{attribute 'GeneratedUsingTerminal: EP2339-0021-0016'}
{attribute addProperty BoxType "EP2339-0021-0016"}
{attribute addProperty Id "Channel_1AT %I*Channel_830843C11Channel_2AT %I*Channel_830843C11Channel_3AT %I*Channel_830843C11Channel_4AT %I*Channel_830843C11Channel_5AT %I*Channel_830843C11Channel_6AT %I*Channel_830843C11Channel_7AT %I*Channel_830843C11Channel_8AT %I*Channel_830843C11Channel_9AT %I*Channel_830843C11Channel_10AT %I*Channel_830843C11Channel_11AT %I*Channel_830843C11Channel_12AT %I*Channel_830843C11Channel_13AT %I*Channel_830843C11Channel_14AT %I*Channel_830843C11Channel_15AT %I*Channel_830843C11Channel_16AT %I*Channel_830843C11Channel_1_1AT %Q*Channel_42CA91F71Channel_2_1AT %Q*Channel_42CA91F71Channel_3_1AT %Q*Channel_42CA91F71Channel_4_1AT %Q*Channel_42CA91F71Channel_5_1AT %Q*Channel_42CA91F71Channel_6_1AT %Q*Channel_42CA91F71Channel_7_1AT %Q*Channel_42CA91F71Channel_8_1AT %Q*Channel_42CA91F71Channel_9_1AT %Q*Channel_42CA91F71Channel_10_1AT %Q*Channel_42CA91F71Channel_11_1AT %Q*Channel_42CA91F71Channel_12_1AT %Q*Channel_42CA91F71Channel_13_1AT %Q*Channel_42CA91F71Channel_14_1AT %Q*Channel_42CA91F71Channel_15_1AT %Q*Channel_42CA91F71Channel_16_1AT %Q*Channel_42CA91F71WcStateAT %I*WcState_9091E0EB2InfoDataAT %I*InfoData_07DD5D1A2"}
{attribute addProperty CRC "2006061753"}
{attribute addProperty Size "36"}
TYPE EP2339_779212B9 EXTENDS EtcSlaveTerminalBase_947E5A46 :
STRUCT
	{attribute addProperty Name "Channel_1"}
	Channel_1 : Channel_830843C1;
	{attribute addProperty Name "Channel_2"}
	Channel_2 : Channel_830843C1;
	{attribute addProperty Name "Channel_3"}
	Channel_3 : Channel_830843C1;
	{attribute addProperty Name "Channel_4"}
	Channel_4 : Channel_830843C1;
	{attribute addProperty Name "Channel_5"}
	Channel_5 : Channel_830843C1;
	{attribute addProperty Name "Channel_6"}
	Channel_6 : Channel_830843C1;
	{attribute addProperty Name "Channel_7"}
	Channel_7 : Channel_830843C1;
	{attribute addProperty Name "Channel_8"}
	Channel_8 : Channel_830843C1;
	{attribute addProperty Name "Channel_9"}
	Channel_9 : Channel_830843C1;
	{attribute addProperty Name "Channel_10"}
	Channel_10 : Channel_830843C1;
	{attribute addProperty Name "Channel_11"}
	Channel_11 : Channel_830843C1;
	{attribute addProperty Name "Channel_12"}
	Channel_12 : Channel_830843C1;
	{attribute addProperty Name "Channel_13"}
	Channel_13 : Channel_830843C1;
	{attribute addProperty Name "Channel_14"}
	Channel_14 : Channel_830843C1;
	{attribute addProperty Name "Channel_15"}
	Channel_15 : Channel_830843C1;
	{attribute addProperty Name "Channel_16"}
	Channel_16 : Channel_830843C1;
	{attribute addProperty Name "Channel_1_1"}
	Channel_1_1 : Channel_42CA91F7;
	{attribute addProperty Name "Channel_2_1"}
	Channel_2_1 : Channel_42CA91F7;
	{attribute addProperty Name "Channel_3_1"}
	Channel_3_1 : Channel_42CA91F7;
	{attribute addProperty Name "Channel_4_1"}
	Channel_4_1 : Channel_42CA91F7;
	{attribute addProperty Name "Channel_5_1"}
	Channel_5_1 : Channel_42CA91F7;
	{attribute addProperty Name "Channel_6_1"}
	Channel_6_1 : Channel_42CA91F7;
	{attribute addProperty Name "Channel_7_1"}
	Channel_7_1 : Channel_42CA91F7;
	{attribute addProperty Name "Channel_8_1"}
	Channel_8_1 : Channel_42CA91F7;
	{attribute addProperty Name "Channel_9_1"}
	Channel_9_1 : Channel_42CA91F7;
	{attribute addProperty Name "Channel_10_1"}
	Channel_10_1 : Channel_42CA91F7;
	{attribute addProperty Name "Channel_11_1"}
	Channel_11_1 : Channel_42CA91F7;
	{attribute addProperty Name "Channel_12_1"}
	Channel_12_1 : Channel_42CA91F7;
	{attribute addProperty Name "Channel_13_1"}
	Channel_13_1 : Channel_42CA91F7;
	{attribute addProperty Name "Channel_14_1"}
	Channel_14_1 : Channel_42CA91F7;
	{attribute addProperty Name "Channel_15_1"}
	Channel_15_1 : Channel_42CA91F7;
	{attribute addProperty Name "Channel_16_1"}
	Channel_16_1 : Channel_42CA91F7;
	{attribute addProperty Name "WcState"}
	WcState : WcState_9091E0EB;
	{attribute addProperty Name "InfoData"}
	InfoData : InfoData_07DD5D1A;
END_STRUCT
END_TYPE

(* stored: Version 1.2.0.0, ProductVersion 3.1.4024.9
   DUT EP2339_779212B9: Id {a7523199-4b1d-47ce-9cd1-b1ab2b94baab} *)
